Staubli VAL3: onF7Event.pgx

program onF7Event()
  local string l_sSwap
  local num l_nResult
  local string l_sMessage
  local string l_sMessage2
  local bool l_bYes
  local string l_sButton[2]
begin
//  // look if the bButton is enable
//  if bButton[6]
//    //
//    // delete a Trajectory
//    //
//    call deleteItem(l_bYes)
//    if l_bYes
//      call trajType:delete(sEvent,l_nResult)
//      if l_nResult==0
//        logMsg("[KERNEL] INTERFACE:Delete the trajectory: "+saveData:sTrajTypeUsing+" "+sEvent)
//        call buildList()
//      else
//        popUpMsg("error code: "+toString("",l_nResult))
//        logMsg("[KERNEL] INTERFACE:Delete the trajectory: "+saveData:sTrajTypeUsing+" "+sEvent+"error code: "+toString("",l_nResult))
//      endIf
//    endIf
//  endIf
end
